FUNCTION_BLOCK StopTask EXTENDS TcoCore.TcoTask IMPLEMENTS IAxisIAI
VAR
    {attribute addProperty Name "<#Deceleration#>"}
    _deceleration : UINT;
END_VAR


IF Execute() THEN
    DriveRef.PlcToDrive.ControlSignal.STP := TRUE;
    DriveRef.PlcToDrive.ControlSignal.RES := TRUE;

    DoneWhen(DriveRef.AxisStatus.NotMoving);
    ThrowWhen(DriveRef.AxisStatus.Error);
END_IF

PROPERTY DriveRef : REFERENCE TO AxisIAI
GET
VAR
    _drive : POINTER TO AxisIAI;
END_VAR
IF __QUERYPOINTER(THIS^._ParentObject, _drive) THEN
    DriveRef REF= _drive^;
END_IF
END_GET
END_PROPERTY

METHOD PUBLIC FB_init : BOOL
VAR_INPUT
    bInitRetains : BOOL; // if TRUE, the retain variables are initialized (warm start / cold start)
    bInCopyCode  : BOOL; // if TRUE, the instance afterwards gets moved into the copy code (online change)
    ParentObject : ITcoObject;
END_VAR
SUPER^.FB_init(bInitRetains := bInitRetains, bInCopyCode := bInCopyCode, ParentObject := ParentObject);
END_METHOD

METHOD INTERNAL InvokeWithParams : ITcoTaskStatus
VAR_INPUT
    inDeceleration : UINT;
END_VAR
_deceleration    := inDeceleration;
InvokeWithParams := THIS^.Invoke();
END_METHOD

(*~
    <docu>
        <summary>
            Executes when task reaches the ```Done``` state .
        </summary>
    </docu>
~*)
METHOD PROTECTED OnDone
DriveRef.PlcToDrive.ControlSignal.STP := FALSE;
DriveRef.PlcToDrive.ControlSignal.RES := FALSE;
DriveRef.Restore();
END_METHOD

(*~
    <docu>
        <summary>
            Restores this instance to the Ready state. Can be called explicitly or from within one of the restore mechanisms.
            <para>
                See also <see cref="PlcDocu.TcoCore.TcoTask.AutoRestorable()"/>
            </para>
        </summary>
    </docu>
~*)
METHOD Restore : ITcoRestorable
SUPER^.Restore();
DriveRef.PlcToDrive.ControlSignal.STP := FALSE;
DriveRef.PlcToDrive.ControlSignal.RES := FALSE;
//DriveRef.Restore();
END_METHOD

END_FUNCTION_BLOCK

(* stored: Version 1.1.0.1, ProductVersion 3.1.4024.12
   POU StopTask: Id {b4ef30fa-ed6d-4bf8-ba5d-3f302d7c811f}, SpecialFunc None
   Property DriveRef: Id {5b3ff870-2b55-4c31-9461-2e97829e64f9}
   Get Get: Id {b801e818-3288-48fe-be97-0dc9bbecfb21}
   Method FB_init: Id {a01b545c-772e-4481-867f-ad7c345a495a}
   Method InvokeWithParams: Id {0033654d-54a2-4d10-b22d-7fa9d28ea5bb}
   Method OnDone: Id {6abf43e7-7dcd-4ca9-9b18-569cf705a015}
   Method Restore: Id {a0cf89d1-51a6-41c5-812c-4927e2dbc215} *)
